PROGRAM MAIN
VAR
	//Elevator:FB_Elevator;
	//Floors:ARRAY[1..4]	OF	ST_Floor;
	State: E_States;
	i: INT;
	//RequestedFloor: INT;
	//ActualFloor: INT;
	Trigger:ARRAY[1..4]	OF	R_TRIG;
END_VAR

CASE	State	OF
	E_States.Call:
		FOR	i:=1	TO	4	DO
			IF	Floors[i].Call	THEN
				RequestedFloor:=i;
			END_IF
		END_FOR
		
		IF	RequestedFloor>ActualFloor	THEN
			State:=E_States.MoveUp;	
		ELSIF	RequestedFloor<ActualFloor	THEN
			State:=E_States.MoveDown;	
		END_IF
	E_States.MoveUp:
		Elevator.MoveUp();
		FOR	i:=1	TO	4	DO
			Trigger[i](clk:=Floors[i].Low);
			IF	Trigger[i].Q	THEN
				ActualFloor:=ActualFloor+1;
			END_IF
		END_FOR
		
		IF	ActualFloor=RequestedFloor	THEN
			State:=E_States.SlowDown;
		END_IF
	E_States.MoveDown:
		Elevator.MoveDown();
		FOR	i:=1	TO	4	DO
			Trigger[i](clk:=Floors[i].High);
			IF	Trigger[i].Q	THEN
				ActualFloor:=ActualFloor-1;
			END_IF
		END_FOR
		
		IF	ActualFloor=RequestedFloor	THEN
			State:=E_States.SlowDown;
		END_IF
		
	E_States.SlowDown:
		Elevator.SlowDown();
		FOR	i:=1	TO	4	DO
			IF	Floors[i].Mid	THEN
				State:=E_States.Stop;
			END_IF
		END_FOR
	E_States.Stop:
		Elevator.Stop();
		State:=E_States.Call;
END_CASE

END_PROGRAM

(* stored: Version 1.1.0.1, ProductVersion 3.1.4024.11
   POU MAIN: Id {437c88b0-71cb-4e07-9d72-857c04460bf1}, SpecialFunc None *)
